FUNCTION_BLOCK FB_DoorOpenClose
VAR_INPUT
	_n									: INT; // array number of which 10 commands to be processed
	_bLock								: BOOL; // 0: Execute unlock command, 1: Execute lock command
	_bFrontDoor							: BOOL;
END_VAR

VAR_OUTPUT
END_VAR

VAR_IN_OUT
END_VAR

VAR
	bErr								: BOOL; // var for error flag
	start								: BOOL;
	_isFrontDoor						: BOOL;
	_bDoorRecoveryStart					: BOOL;
	_DoorOpen_Permissive				: BOOL;
	
	iStep								: INT	:= 1;
	_iLevel								: INT;

	iSendEvent							: UINT	:= 1;
	
	sStatus								: STRING; // var for error message
	sLogName							: STRING;
	sFailReason							: STRING;
	sModuleID							: STRING;
	_eFailLogName						: STRING;
	_ePassLogName						: STRING;
	
	tim									: TON;
	timDwrUp							: TON;
	timDoorRecStartDel					: TON;
	
	rtStart								: R_TRIG;
	
	EmptyEvents							: ST_Event;
	CmdEmpty							: ST_Command;
	requestedState						: E_State	:= E_State.eEnabled;
	eEventName							: E_EventName;
	_eFailEvent							: E_EventName;
	_ePassEvent							: E_EventName;
	stMultiLevelVIO						: ST_TCMultiLevel_VIO;
	_arrRCMD							: ARRAY [1..NO_OF_CMD_BUFFER] OF ST_Command;
	_arrEvent							: ARRAY [1..NO_OF_EVENT_BUFFER] OF ST_Event;
	//fbCmdAndEventUpdate: FB_CmdAndEventUpdate;
	_sanityCheck						: INT;
END_VAR

rtStart(CLK := start , Q=> );
IF rtStart.Q THEN
	iStep																			:= 1;
END_IF

IF (NOT start) THEN
	RETURN;
END_IF


///////////////////////////////////////////////////////////////////////////////////////////////////////////////////////////////////////////////////////////////////////////////
//	State machine
///////////////////////////////////////////////////////////////////////////////////////////////////////////////////////////////////////////////////////////////////////////////

CASE iStep OF
	0: (*Idle*)
		;
		
	1: (*Reset*)
	
		(*Action*)
		tim(IN := FALSE);
		timDwrUp(IN := FALSE);
		iStep																		:= 2; // Sanity Check
	
	2:	
		(*Action*)
		sStatus																		:= '';
		bErr																		:= FALSE;
		stMultiLevelVIO 															:= arrTCMultiLevel[_iLevel].fbTCMultiLevelSeq.P_stTCMultiLevelVIO;

		
///////////////////////////////////////////////////////////////////////////////////////////////////////////////////////////////////////////////////////////////////////////////
//	Door Unlock
///////////////////////////////////////////////////////////////////////////////////////////////////////////////////////////////////////////////////////////////////////////////
		IF (NOT _bLock) THEN
//Front Door
			IF _bFrontDoor THEN
				(*Sanity Check*)
				(*_sanityCheck		:= arrTCMultiLevel[_iLevel].fbTCMultiLevelSeq.M_IsSanityCheckFailed(stMultiLevelVIO:= stMultiLevelVIO, sMsg=> sStatus);
				IF  _sanityCheck <> 0 THEN
					bErr												:= TRUE;
					ALMTC.Level[_iLevel].AlarmID[_sanityCheck]			:= TRUE;
					iStep												:= 20;
				END_IF
				
				IF ALMTC.Level[_iLevel].AlarmID[E_AlarmID.APIsNotInUPPosition] THEN
					bErr												:= TRUE;
					sStatus												:= 'AP is not Deactuated (UP)';
					iStep												:= 20;
				ELSIF ALMTC.Level[_iLevel].AlarmID[E_TIIAlarm.ipAPReady] THEN
					bErr												:= TRUE;
					sStatus												:= 'AP is not Ready';
					iStep												:= 20;
				END_IF
				*)
				(*IF (NOT bErr) THEN
					arrTCMultiLevel[_iLevel].stGblParam.bDrawerUpBefFrtDoorOpen		:= TRUE;
					arrTCMultiLevel[_iLevel].fbTCMultiLevelSeq.P_stParam 			:= arrTCMultiLevel[_iLevel].stGblParam;
					iStep															:= 4; // Trigger door output
				END_IF*)
				
				////////////////////////////////////// I MOVED OPEN FRONT DOOR TO SEQUENCE BECAUSE OF ALL HERE RUBBISH CODE////////////////////////////////////////////////////
				start																	:= FALSE;
				arrTCMultiLevel[_iLevel].stGblParam.bDrawerUpBefFrtDoorOpen				:= TRUE;
				RETURN;
				////////////////////////////////////// I MOVED OPEN FRONT DOOR TO SEQUENCE BECAUSE OF THIS RUBBISH CODE////////////////////////////////////////////////////
//Back Door
			ELSE
				IF (NOT bErr) THEN
					
					stMultiLevelVIO.opCellDoorClosed 								:= _bLock;
					arrTCMultiLevel[_iLevel].fbTCMultiLevelSeq.P_stTCMultiLevelVIO 	:= stMultiLevelVIO;
					iStep															:= 20; // Set event
					//END_IF
				END_IF
			END_IF
		
///////////////////////////////////////////////////////////////////////////////////////////////////////////////////////////////////////////////////////////////////////////////
//	Door Lock
///////////////////////////////////////////////////////////////////////////////////////////////////////////////////////////////////////////////////////////////////////////////
		ELSE
//FRONT DOOR
			IF _bFrontDoor THEN
				
				// Make sure front door is closed
				IF (NOT stMultiLevelVIO.ipTCCellTbotSideDoorOpenCloseStatus01) OR (NOT stMultiLevelVIO.ipTCCellTbotSideDoorOpenCloseStatus02) THEN
					bErr															:= TRUE;
					sStatus															:= 'Front Door is not Closed';
					iStep															:= 20; // Set event
				END_IF
				
				IF (NOT bErr) THEN
					//Lock the Door (on the actual output)
					stMultiLevelVIO 												:= arrTCMultiLevel[_iLevel].fbTCMultiLevelSeq.P_stTCMultiLevelVIO;
					stMultiLevelVIO.opCellTBOtSideDoorClosed1 						:= _bLock;
					stMultiLevelVIO.opCellTBOtSideDoorClosed2 						:= _bLock;
					arrTCMultiLevel[_iLevel].fbTCMultiLevelSeq.P_stTCMultiLevelVIO 	:= stMultiLevelVIO;
					tim(IN:=TRUE,PT:=T#1000MS);
					
					IF tim.Q THEN
						stMultiLevelVIO 											:= arrTCMultiLevel[_iLevel].fbTCMultiLevelSeq.P_stTCMultiLevelVIO;
						
						IF NOT (stMultiLevelVIO.ipTCCellTbotSideDoorLocked01 AND stMultiLevelVIO.ipTCCellTbotSideDoorLocked02) THEN
							bErr													:= TRUE;
							sStatus													:= 'Door Lock Error, Front Door Lock Status not Detected After Door Lock Activated';
							iStep													:= 20; // Set event
						ELSE
							arrTCMultiLevel[_iLevel].stGblParam.bDoorClose			:= SEL(_bLock,FALSE,TRUE);
							arrTCMultiLevel[_iLevel].fbTCMultiLevelSeq.P_stParam 	:= arrTCMultiLevel[_iLevel].stGblParam;
								//timDoorRecStartDel(IN:=FALSE);
								_bDoorRecoveryStart 								:= TRUE;
								iStep												:= 3; // Spare
								bErr												:= FALSE;
						END_IF	
						
						tim(IN:= FALSE);
					END_IF
				END_IF
			
//BACK DOOR
			ELSE 
				// Make sure back door is closed
				IF (NOT stMultiLevelVIO.ipTCCellDoorOpenCloseStatus) THEN
					bErr															:= TRUE;
					IF bDebugCart THEN 
						sStatus														:= 'Cell Door is not Closed (Back)';
					ELSE
						sStatus														:= 'Cell Door is not Closed !!';
					END_IF
					iStep															:= 20; // Set event
				END_IF
				
				IF (NOT bErr) THEN 
					stMultiLevelVIO.opCellDoorClosed 								:= _bLock;
					arrTCMultiLevel[_iLevel].fbTCMultiLevelSeq.P_stTCMultiLevelVIO 	:= stMultiLevelVIO;
					tim(IN:= TRUE, PT:= T#1000MS);
					
					IF tim.Q THEN
						stMultiLevelVIO 											:= arrTCMultiLevel[_iLevel].fbTCMultiLevelSeq.P_stTCMultiLevelVIO;
						
						IF (NOT stMultiLevelVIO.ipTCCellDoorClosed) THEN
							bErr																:= TRUE;
							sStatus																:= 'Door Lock Error, Door LockStatus not ON After Door Lock';
							iStep																:= 20; // Set event
						ELSE
							arrTCMultiLevel[_iLevel].stGblParam.bDoorClose			:= SEL(_bLock,FALSE,TRUE);
							arrTCMultiLevel[_iLevel].fbTCMultiLevelSeq.P_stParam 	:= arrTCMultiLevel[_iLevel].stGblParam;
							
							IF _bLock THEN
								_bDoorRecoveryStart 								:= TRUE;
								iStep												:= 3; // Spare
								bErr												:= FALSE;	
								
							END_IF
						END_IF	
						tim(IN:= FALSE);
					END_IF
				END_IF
			END_IF	
		END_IF
		
	3: (*Spare*)
		
		(*Transition*)
		iStep																		:= 20;
		
	20: (*Set event*)

		(*Action*)
		IF bErr THEN
			eEventName																:= _eFailEvent;
			sLogName																:= _eFailLogName;
		ELSE
			eEventName																:= _ePassEvent;
			sLogName																:= _ePassLogName;
		END_IF
		
		sFailReason																	:= sStatus;
		
		CmdAndEventProcess.fbCmdAndEventUpdate.M_AddEvent(
			sLogName																:= sLogName, 
			eEventName																:= eEventName, 
			eModuleID																:= _arrRCMD[_n].eModuleID, 
			iParam																	:= _arrRCMD[_n].iParam,
			sParam																	:= _arrRCMD[_n].sParam, 
			bParam																	:= _arrRCMD[_n].bParam, 
			dParam																	:= _arrRCMD[_n].dParam,
			sFailReason																:= sFailReason);
		
		start																		:= FALSE;
		IF _bDoorRecoveryStart THEN
			arrTCMultiLevel[_iLevel].stGblParam.bDoorRecoveryStarted				:= TRUE;
			arrTCMultiLevel[_iLevel].stGblParam.stDoorRecovEvnt.sLogName			:= 'DoorRecoveryStarted';
			arrTCMultiLevel[_iLevel].stGblParam.stDoorRecovEvnt.eEventName			:= E_EventName.DoorRecoveryStarted;
			arrTCMultiLevel[_iLevel].stGblParam.stDoorRecovEvnt.eModuleID			:= _arrRCMD[_n].eModuleID;
			arrTCMultiLevel[_iLevel].fbTCMultiLevelSeq.P_stParam					:= arrTCMultiLevel[_iLevel].stGblParam;
			timDoorRecStartDel(IN:= FALSE);
			_bDoorRecoveryStart														:= FALSE;
		END_IF
		
		(*Transition*)
		iStep																		:= 0; // Idle
END_CASE

METHOD Execute : BOOL
VAR_INPUT
	n											: INT;
	iLevel										: INT;
	bLock										: BOOL;
	bFrontDoor									: BOOL;
	eFailEvent									: E_EventName;
	ePassEvent									: E_EventName;
	eFailLogName								: STRING;
	ePassLogName								: STRING;
END_VAR

VAR_IN_OUT
	arrRCMD										: ARRAY [1..NO_OF_CMD_BUFFER] OF ST_Command;
	arrEvent									: ARRAY [1..NO_OF_EVENT_BUFFER] OF ST_Event;
END_VAR
start												:= TRUE;
_arrRCMD											:= arrRCMD;
_arrEvent											:= arrEvent;
_ilevel												:= SEL(ilevel>100, ilevel, ilevel-100);
_bFrontDoor											:= SEL(ilevel>100, FALSE, TRUE);
_bLock												:= bLock;
_bFrontDoor											:= bFrontDoor;
_n													:= n;
_eFailEvent											:= eFailEvent ;
_ePassEvent											:= ePassEvent;
_eFailLogName										:= eFailLogName;
_ePassLogName										:= ePassLogName;
END_METHOD

METHOD Reset : BOOL
VAR_INPUT
END_VAR
start:=false;
END_METHOD

END_FUNCTION_BLOCK

(* stored: Version 1.1.0.1, ProductVersion 3.1.4022.18
   POU FB_DoorOpenClose: Id {cc9007dd-01c7-4c39-b58e-94433c500190}, SpecialFunc None
   Method Execute: Id {ca3b77b5-2a99-4c78-99c2-1d04539e022e}
   Method Reset: Id {556c6df1-3e10-4114-8292-b48bc44863e3} *)
